RoboDK station: Test_paint.rdk

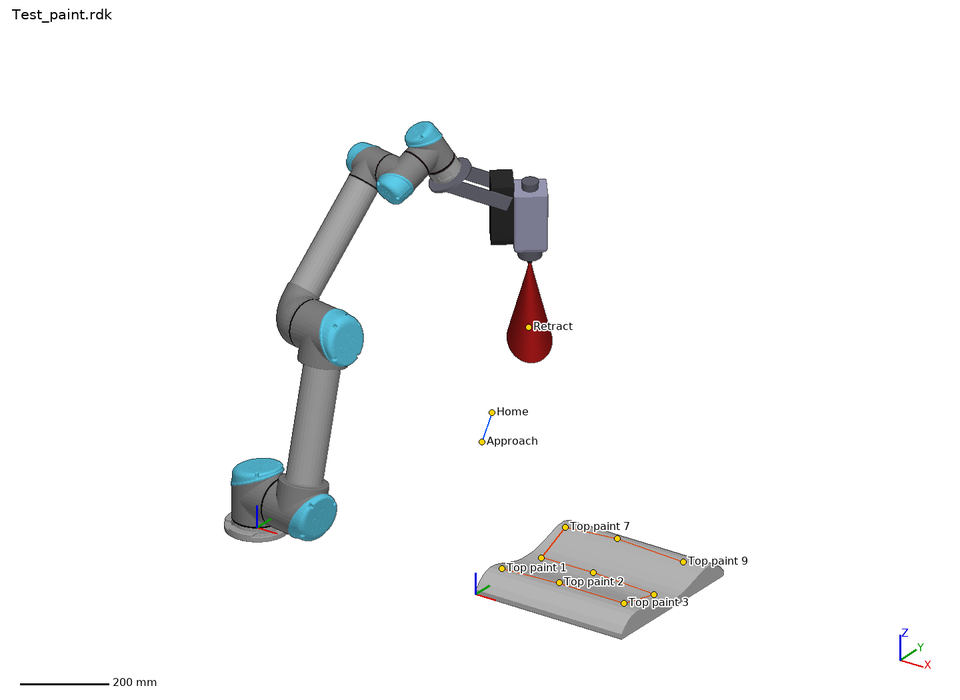
[picture v0: the station drawn from its stored meshes, robots at their saved joint values, targets as dots, program paths as lines]
Station Test_paint (saved by RoboDK 5.6.3). Poses are relative to the parent item; angles as X-Y-Z fixed-axis rotations.
  - frame UR5 Base at (-510, 500, 100) mm
    - robot UR5: 6 axes
        modified DH rows (alpha deg, a mm, theta deg, d mm): 0, 0, 0, 89.2; 90, 0, 180, 0; 0, 425, 0, 0; 0, 392, 0, 109.3; -90, 0, 0, 94.75; 90, 0, 0, 82.5
        joint limits [-360, -360, -360, -360, -360, -360] to [360, 360, 360, 360, 360, 360]; home [0, -90, -90, 0, 90, 0]; saved at [79.297, -101.992, -30.383, -110.251, 75.25, 128.896]
      - tool Paint gun, TCP at (50, 0, 450) mm, rotated rx 0 ry 30 rz 0 deg, size 203.2 x 279.7 x 471.5 mm
  - frame Frame 2 at (90, 500, 100) mm
    - object Object Inspection at (0, 0, 0) mm, size 400 x 400 x 46.2 mm, geometry from Object Inspection.stp
    - target Home (Cartesian target) at (222.6, -255.47, 619.13) mm, rotated rx -173.89 ry 49.82 rz -169.63 deg; joints [-29.118, -94.632, -62.04, -35.352, 123.53, 79.29] of UR5
    - target Approach (Cartesian target) at (10, 10, 380) mm, rotated rx -180 ry 0 rz -180 deg; joints [17.877, -96.365, -31.623, -113.224, 81.171, 105.607] of UR5
    - target Retract (Cartesian target) at (-269.88, 591.52, 355.8) mm, rotated rx 173.53 ry 0.2 rz -141.48 deg; joints [231.19, -47.742, -32.05, -41.019, -90.865, 104.162] of UR5
    - target Top paint 1 (Cartesian target) at (25, 65.9, 45.8) mm, rotated rx 178.04 ry -0.03 rz -180 deg; joints [171.337, -2.928, -104.386, -12.167, -83.999, 83.442] of UR5
    - target Top paint 2 (Cartesian target) at (170, 83.5, 43.12) mm, rotated rx 167.91 ry -1 rz -179.89 deg; joints [166.727, -0.021, -84.799, -31.866, -73.215, 83.979] of UR5
    - target Top paint 3 (Cartesian target) at (350, 81.72, 43.5) mm, rotated rx -167.91 ry 1 rz -179.89 deg; joints [185.823, -8.26, -45.588, -66.678, -103.405, 88.891] of UR5
    - target Top paint 4 (Cartesian target) at (350, 198.77, 18.33) mm, rotated rx 179.51 ry 0 rz -180 deg; joints [186.633, -8.042, -43.892, -67.942, -92.886, 95.995] of UR5
    - target Top paint 5 (Cartesian target) at (175, 212.13, 18.42) mm, rotated rx 179.51 ry 0 rz -180 deg; joints [189.963, 2.259, -81.565, -40.381, -94.541, 98.891] of UR5
    - target Top paint 6 (Cartesian target) at (35, 208.03, 18.39) mm, rotated rx -179.51 ry 0 rz 180 deg; joints [193.609, 2.53, -100.87, -20.87, -97.174, 101.605] of UR5
    - target Top paint 7 (Cartesian target) at (20, 323.03, 44.54) mm, rotated rx -168.03 ry -0.98 rz 179.9 deg; joints [215.564, -2.325, -78.558, -27.821, -115.398, 118.103] of UR5
    - target Top paint 8 (Cartesian target) at (150, 339.98, 46) mm, rotated rx 178.04 ry -0.03 rz -180 deg; joints [201.339, -2.481, -72.564, -43.765, -98.869, 109.582] of UR5
    - target Top paint 9 (Cartesian target) at (340, 327.93, 45.59) mm, rotated rx 178.04 ry -0.03 rz -180 deg; joints [195.425, -17.564, -25.462, -76.457, -95.987, 104.374] of UR5
  - program Apprachmove (4 instructions, listed below)
  - program PaintTop (11 instructions, listed below)
  - program Retract (3 instructions, listed below)
  - program MainProgram (5 instructions, listed below)
  - Python program SprayOn (listed below)
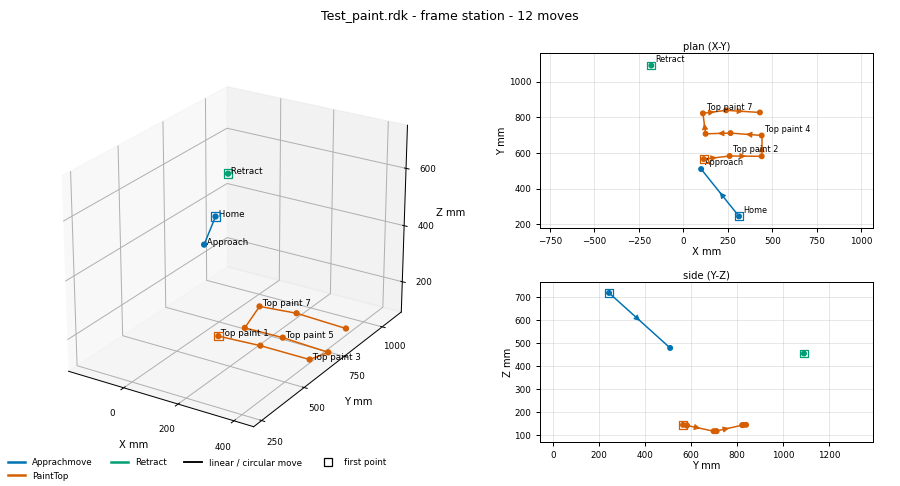
[picture p0: tool path of Test_paint.rdk in frame station, 12 of 12 moves have a stored position in this frame; points joined in program order, loops and branches not executed]

--- program Apprachmove (robot UR5) ---
  Set Ref.: Frame 2
  Set Tool: Paint gun
  MoveL (Home)
  MoveL (Approach)

--- program PaintTop (robot UR5) ---
  Set Ref.: Frame 2
  Set Tool: Paint gun
  MoveL (Top paint 1)
  MoveL (Top paint 2)
  MoveL (Top paint 3)
  MoveL (Top paint 4)
  MoveL (Top paint 5)
  MoveL (Top paint 6)
  MoveL (Top paint 7)
  MoveL (Top paint 8)
  MoveL (Top paint 9)

--- program Retract (robot UR5) ---
  Set Ref.: Frame 2
  Set Tool: Paint gun
  MoveL (Retract)

--- program MainProgram (robot UR5) ---
  Call Apprachmove
  Call SprayOn(1)
  Call PaintTop
  Call SprayOn(0)
  Call Retract

--- Python program SprayOn ---
# This macro allows simulating a spray gun for painting or to simulate the trace of inspaction
#
# You can call SprayOn(1) to simulate turning the Spray gun ON or SprayOn(0) to stop simulating the gun
# Calling SprayOn(-1) clears all displayed data
# The macro will output spray gun statistics
#
# --------------------------------------------------------------
# This script shows how to create "spray" object in RoboDK that allows simulating particle deposition by using:
# RDK.Spray_Add(tool, object, options_command, volume, geometry)
#    tool: tool item (TCP) to use
#    object: object to project the particles
#    options_command (optional): string to specify options.
#    volume (optional): Matrix of parameters defining the volume of the spray gun
#    geometry (optional): Matrix of vertices defining the triangles.
#
# More information here:
# https://robodk.com/doc/en/PythonAPI/robodk.html#robodk.robolink.Robolink.Spray_Add
# https://robodk.com/doc/en/RoboDK-API.html
#
# The scripts ArcStart, ArcEnd and WeldOn and SpindleOn behave in a similar way, the only difference is the default behavior
# This behavior simmulates Fanuc Arc Welding and triggers appropriate output when using the customized post processor.
# Select ESC to clear the trace manually.
#
# Example scripts that use Spray_Add:
#     SpindleOn / SpindleOff    -> Turn trace On/Off
#     ArcOn / ArcOff            -> Turn trace On/Off
#     SprayOn / SprayOff        -> Simulate a spray given a workspace volume (for painting)
#     WeldOn / WeldOff          -> Support for multiple weld guns

#------------------------------------------------------------------

# Use a specific tool as a spray gun
Tool_Name = None
#Tool_Name = 'Tool 2'

# Use a specific object to project particles:
Object_Name = None
#Object_Name = 'Part'

# Define the default action (0 to deactivate, +1 to activate, -1 to clear any spray gun simulation)
# Setting it to None will display a message
ACTION = None

from robodk.robolink import *  # API to communicate with RoboDK
from robodk.robomath import *  # basic matrix operations
from robodk.robodialogs import *

RDK = Robolink()

# quit if we are not in simulation mode
if RDK.RunMode() != RUNMODE_SIMULATE:
    quit()

# Get any previously added spray gun simulations and display statistics (spray on the part vs spray falling out of the part)
info, data = RDK.Spray_GetStats()
if data.size(1) > 0:
    print("Spray gun statistics:")
    print(info)
    print(data.tr())
    # # Diplay statistics
    # RDK.ShowMessage("Material used: %.1f%%<br>Material waisted: %.1f%%<br>Total particles: %.1f" % (data[1,0],data[2,0],data[3,0]), True)
    # # Clear previous spray
    # RDK.Spray_Clear()

# Check if we are running this program inside another program and passing arguments
import sys
if len(sys.argv) > 1:
    ACTION = int(sys.argv[1])

# If the default ACTION is None, display a message to activate/deactivate the spray gun
if ACTION is None:
    print('Note: This macro can be called as Spray(1) or SprayOn(0)')
    entry = mbox('Turn gun ON or OFF', ('On', '1'), ('Off', '0'))
    if not entry:
        quit()
    ACTION = int(entry)

if ACTION == 0:
    # Turn the gun off
    RDK.Spray_SetState(SPRAY_OFF)

elif ACTION < 0:
    # Clear all spray simulations (same as pressing ESC key)
    RDK.Spray_Clear()

elif ACTION > 0:
    # Create a new spray gun object in RoboDK
    # by using RDK.Spray_Add(tool, object, options_command, volume, geometry)
    # tool: tool item (TCP) to use
    # object: object to project the particles
    # options_command (optional): string to specify options. Example:
    #     STEP=AxB: Defines the grid to be projected 1x1 means only one line of particle projection (for example, for welding)
    #     PARTICLE: Defines the shape and size of particle (sphere or particle), unless a specific geometry is provided:
    #       a- SPHERE(radius, facets)
    #       b- SPHERE(radius, facets, scalex, scaley, scalez)
    #       b- CUBE(sizex, sizey, sizez)
    #     RAND=factor: Defines a random factor factor 0 means that the particles are not deposited randomly
    #     ELLYPSE: defines the volume as an ellypse (default)
    #     RECTANGLE: defines the volume as a rectangle
    #     PROJECT: project the particles to the surface (default) (for welding, painting or scanning)
    #     NO_PROJECT: does not project the particles to the surface (for example, for 3D printing)
    #
    # volume (optional): Matrix of parameters defining the volume of the spray gun
    # geometry (optional): Matrix of vertices defining the triangles.

    tool = 0  # auto detect active tool
    obj = 0  # auto detect object in active reference frame
    if Tool_Name is not None:
        tool = RDK.Item(Tool_Name, ITEM_TYPE_TOOL)

    if Object_Name is not None:
        obj = RDK.Item(Object_Name, ITEM_TYPE_OBJECT)
    # We can specify a given tool object and/or object
    #robot = RDK.Item("ABB IRB 2600-12/1.85", ITEM_TYPE_ROBOT)
    #tools = robot.Childs()
    #if len(tools) > 0:
    #    tool = tools[0]
    #obj = RDK.Item('object', ITEM_TYPE_OBJECT)

    options_command = "ELLYPSE PROJECT PARTICLE=SPHERE(4,8,1,1,0.5) STEP=8x8 RAND=2"  # simulate
    #options_command = "PARTICLE=CUBE(10,10,2) STEP=8x8"
    #options_command = "PARTICLE=SPHERE(4,8) STEP=8x8"
    #options_command = "PARTICLE=SPHERE(4,8,1,1,0.1) STEP=8x8 RAND=3"

    # Example commands for welding:
    # options_command = "PROJECT PARTICLE=SPHERE(4,8)"
    # options_command = PARTICLE=SPHERE(4,8) STEP=1x0

    # define the ellypse volume as p0, pA, pB, colorRGBA (close and far), in mm
    # coordinates must be provided with respect to the TCP
    close_p0 = [0, 0, -200]  # xyz in mm: Center of the conical ellypse (side 1)
    close_pA = [5, 0, -200]  # xyz in mm: First vertex of the conical ellypse (side 1)
    close_pB = [0, 10, -200]  # xyz in mm: Second vertex of the conical ellypse (side 1)
    close_color = [1, 0, 0, 1]  # RGBA (0-1)

    far_p0 = [0, 0, 50]  # xyz in mm: Center of the conical ellypse (side 2)
    far_pA = [60, 0, 50]  # xyz in mm: First vertex of the conical ellypse (side 2)
    far_pB = [0, 120, 50]  # xyz in mm: Second vertex of the conical ellypse (side 2)
    far_color = [0, 0, 1, 0.2]  # RGBA (0-1)

    close_param = close_p0 + close_pA + close_pB + close_color
    far_param = far_p0 + far_pA + far_pB + far_color
    volume = Mat([close_param, far_param]).tr()
    RDK.Spray_Add(tool, obj, options_command, volume)
    RDK.Spray_SetState(SPRAY_ON)

    # Another example with a varying rectancular shape
    # define the rectangular volume as p0, pA, pB, colorRGBA (close and far)
    # close_param = [-90,-117,  0,  90,-117,0,   -90,117,  0,       0.2,0.2,1,.1]
    # far_param   = [-175,-190,200, 175,-190,200,   -175,190,200,   0.5,0,0,.9]
    # volume = Mat([close_param, far_param])
    # RDK.Spray_Add(tool, obj, "RECTANGLE PARTICLE=SPHERE(2,5) STEP=15x15 RAND=3", volume.tr())
    # RDK.Spray_SetState(SPRAY_ON)

    # Optional: define geometry as a list of triangles with normals (instead of a scaled cube or a sphere)
    # geom = Mat([[0,0,0,   0,0,1], [5,0,0,   0,0,1], [0,5,0,   0,0,1]])
    # RDK.Spray_Add(tool, obj, "STEP=8x8 RANDX=3", volume.tr(), geom.tr())
    # RDK.Spray_SetState(SPRAY_ON)
